// TIA Portal V18 export
FUNCTION "DIadv" : Void   // FC10007, LAD
{ S7_Optimized_Access := 'TRUE' }
VERSION : 0.1
// stored: AutoNumber false, IsIECCheckEnabled false, SetENOAutomatically false, UDAEnableTagReadback false
   VAR_INPUT
      xInput : Bool;
      xInversion : Bool;   // 0-direct / 1-reverse
      cDelayOffSec : Byte;
      cDelayOnSec : Byte;
   END_VAR
   VAR_OUTPUT
      xOutputFiltered : Bool;
      xOutputUnFiltered : Bool;
   END_VAR
   VAR_IN_OUT
      xMemoryOut : Bool;
      xMemoryIn : Bool;
      cMemory : Byte;
      iCounterIn : Int;
      iCounterOut : Int;
   END_VAR
   VAR_TEMP
      xInit : Bool;
      InOut_1 : Bool;
      xTemp : Bool;
   END_VAR
BEGIN

REGION Network 1 (SCL): Ініціалізація
   // --- Ініціалізація на першому циклі ---
   IF #xInit THEN
       #xMemoryIn := #xInput;
       #xTemp := #xInput;
       #xMemoryOut := #xTemp;
       // лічильники залишаємо як є (0 за замовчуванням або з рецепта)
       #xInit := FALSE;
   END_IF;
END_REGION

REGION Network 2 (SCL): Inversion
   IF #xInversion THEN
       #xOutputFiltered := NOT #xInput;
   ELSE
       #xOutputFiltered := #xInput;
   END_IF;
END_REGION

REGION Network 3 (SCL): Затримки на включ/вимкн
   #xOutputUnFiltered := #xInput;
END_REGION

REGION Network 4 (SCL): // --- Підрахунок змін на вході ---
   IF #xInput <> #xMemoryIn THEN
       IF #iCounterIn < 32767 THEN
           #iCounterIn := #iCounterIn + 1;
       ELSE
           #iCounterIn := 0;
       END_IF;
   END_IF;
END_REGION

REGION Network 5 (SCL): // --- Підрахунок змін на виході ---
   IF #xOutputFiltered <> #xMemoryOut THEN
       IF #iCounterOut < 32767 THEN
           #iCounterOut := #iCounterOut + 1;
       ELSE
           #iCounterOut := 0;
       END_IF;
   END_IF;
END_REGION

REGION Network 6 (SCL)
   // --- Оновлення попередніх значень ---
   #xMemoryIn := #xInput;
   #xMemoryOut := #xOutputFiltered;
END_REGION
END_FUNCTION
